(* IEC 61131-3 sources: AXOpen/src/showcase/app/src/core/AXOpen.AxoTask, 4 files *)

(* ---- AxoTaskAbortedExample.st ---- *)
USING AXOpen.Core;

NAMESPACE AxoTaskExamples

    // Demonstrates the Aborted terminal state in AxoTaskView:
    //   - Invoke kicks the task into Busy.
    //   - After a fixed number of Execute cycles, Abort() transitions the
    //     task to Aborted (stop icon + Resume button appear in the view).
    //   - Resume returns the task to Busy; counter is reset on Abort so the
    //     next run gets a fresh window before re-aborting.
    //   - Restore (Reset task button) returns the task to Ready.
    {S7.extern=ReadWrite}
    CLASS AxoTaskAbortedExample EXTENDS AXOpen.Core.AxoObject

        //<ComponentDeclaration>
        VAR PUBLIC
            {#ix-set:AttributeName = "<#Aborting task#>"}
            _abortingTask : AXOpen.Core.AxoTask;
            _counter : ULINT;
        END_VAR
        //</ComponentDeclaration>

        METHOD PUBLIC Execute

            //<Initialization>
            _abortingTask.Run(THIS);
            //</Initialization>

            //<AxoTaskAbortedPattern>
            IF _abortingTask.Execute() THEN
                _counter := _counter + ULINT#1;
                IF _counter > ULINT#250 THEN
                    _counter := ULINT#0;
                    _abortingTask.Abort();
                END_IF;
            END_IF;

            IF _abortingTask.IsReady() THEN
                _counter := ULINT#0;
            END_IF;
            //</AxoTaskAbortedPattern>

        END_METHOD
    END_CLASS
END_NAMESPACE

(* ---- AxoTaskDisabledExample.st ---- *)
USING AXOpen.Core;

NAMESPACE AxoTaskExamples

    // Demonstrates the disabled-state indicator in AxoTaskView:
    //   - The task is kept perpetually Busy (self-invoked, never completed),
    //     so it always sits in an "active" state.
    //   - Rendering this task through a DISABLED / display-only AxoTaskView
    //     (Disable=true, e.g. the Status presentation) draws the activity
    //     circle with a lock icon INSIDE it, instead of replacing the circle.
    //   - Note: a task disabled on the PLC side via SetIsDisabled(TRUE) aborts
    //     while Busy (see AxoTaskLight.Execute), so the lock-inside-circle
    //     visual is a VIEW-level disable of a genuinely running task.
    {S7.extern=ReadWrite}
    CLASS AxoTaskDisabledExample EXTENDS AXOpen.Core.AxoObject

        //<ComponentDeclaration>
        VAR PUBLIC
            {#ix-set:AttributeName = "<#Always-active task — render display-only#>"}
            _activeTask : AXOpen.Core.AxoTask;
            {#ix-set:AttributeName = "<#Idle (Ready) task — render display-only#>"}
            _idleTask : AXOpen.Core.AxoTask;
        END_VAR
        //</ComponentDeclaration>

        METHOD PUBLIC Execute

            //<Initialization>
            _activeTask.Run(THIS);
            _idleTask.Run(THIS);
            //</Initialization>

            //<AxoTaskAlwaysActivePattern>
            // Execute() first (satisfies the cyclic-execute-called check), then
            // Invoke(). Invoke() only acts while the task is Ready, so once the
            // task is Busy it is a no-op and the task stays active indefinitely.
            _activeTask.Execute();
            _activeTask.Invoke();
            //</AxoTaskAlwaysActivePattern>

            //<AxoTaskIdlePattern>
            // _idleTask is wired into the object tree but never invoked, so it
            // stays in the Ready (not-busy) state. Rendered through a disabled
            // view it shows the lock inside the empty Ready circle.
            //</AxoTaskIdlePattern>

        END_METHOD
    END_CLASS
END_NAMESPACE

(* ---- AxoTaskDocuExample.st ---- *)
USING AXOpen.Core;

NAMESPACE AxoTaskExamples
    {S7.extern=ReadWrite}
    CLASS AxoTaskDocuExample EXTENDS  AXOpen.Core.AxoObject
        VAR PUBLIC
            {#ix-set:AttributeName = "<#Task name#>"}
            _myTask : AxoTask;
            _myCounter : ULINT;
        END_VAR

        METHOD PUBLIC Initialize
            // Initialization of the context needs to be called first
            // It does not need to be called cyclically, just once
            _myTask.Run(THIS);
        END_METHOD

        METHOD PUBLIC Execute
            _myTask.Run(THIS);
            // Cyclicall call of the Execute
            IF _myTask.Execute() THEN
                _myCounter := _myCounter + ULINT#1;
                _myTask.DoneWhen(_myCounter = ULINT#100);
            END_IF;
            IF _myTask.IsDone() THEN
                _myCounter := ULINT#0;
            END_IF;
        END_METHOD

        METHOD Examples
        //<AxoTaskInvokeDone>
            IF _myTask.Invoke().IsDone() THEN
                ; //Do something
            END_IF;
        //</AxoTaskInvokeDone>

        //<AxoTaskInvokeDoneSeparatelly>
            _myTask.Invoke();

            IF _myTask.IsDone() THEN
                ; //Do something
            END_IF;
        //</AxoTaskInvokeDoneSeparatelly>

        //<AxoTaskRunning>
             IF _myTask.Invoke().IsBusy() THEN
                ; //Do something
            END_IF;
        //</AxoTaskRunning>

        //<AxoTaskError>
            IF _myTask.Invoke().HasError() THEN
                ; //Do something
            END_IF;
        //</AxoTaskError>

        //<AxoTaskInvoke>
            _myTask.Invoke();
        //</AxoTaskInvoke>
        END_METHOD
    END_CLASS

    //<AxoTaskEventLikeMethods>
    {S7.extern=ReadWrite}
    CLASS MyTaskExample EXTENDS AXOpen.Core.AxoTask
        VAR
            OnAbortCounter : ULINT;
            OnResumeCounter : ULINT;
            OnDoneCounter : ULINT;
            OnErrorCounter : ULINT;
            OnRestoreCounter : ULINT;
            OnStartCounter : ULINT;
            WhileErrorCounter : ULINT;
        END_VAR
        METHOD PROTECTED OVERRIDE OnAbort
            OnAbortCounter := OnAbortCounter + ULINT#1;
        END_METHOD

        METHOD PROTECTED OVERRIDE OnResume
            OnResumeCounter := OnResumeCounter + ULINT#1;
        END_METHOD

        METHOD PROTECTED OVERRIDE OnDone
            OnDoneCounter := OnDoneCounter + ULINT#1;
        END_METHOD

        METHOD PROTECTED OVERRIDE OnError
            OnErrorCounter := OnErrorCounter + ULINT#1;
        END_METHOD

        METHOD PROTECTED OVERRIDE OnRestore
            OnRestoreCounter := OnRestoreCounter + ULINT#1;
        END_METHOD

        METHOD PROTECTED OVERRIDE OnStart
            OnStartCounter := OnStartCounter + ULINT#1;
        END_METHOD

        METHOD PROTECTED OVERRIDE WhileError
            WhileErrorCounter := WhileErrorCounter + ULINT#1;
        END_METHOD
    END_CLASS
    //</AxoTaskEventLikeMethods>
END_NAMESPACE

(* ---- AxoTaskErrorExample.st ---- *)
USING AXOpen.Core;

NAMESPACE AxoTaskExamples

    // Demonstrates the Error terminal state in AxoTaskView:
    //   - Invoke kicks the task into Busy.
    //   - After a fixed number of Execute cycles, ErrorDetails is populated
    //     and ThrowWhen(TRUE) transitions the task to Error.
    //   - Restore (Reset task button) returns the task to Ready and clears
    //     the counter for the next demonstration.
    {S7.extern=ReadWrite}
    CLASS AxoTaskErrorExample EXTENDS AXOpen.Core.AxoObject

        //<ComponentDeclaration>
        VAR PUBLIC
            {#ix-set:AttributeName = "<#Failing task#>"}
            _failingTask : AXOpen.Core.AxoTask;
            _counter : ULINT;
        END_VAR
        //</ComponentDeclaration>

        METHOD PUBLIC Execute

            //<Initialization>
            _failingTask.Run(THIS);
            //</Initialization>

            //<AxoTaskErrorPattern>
            IF _failingTask.Execute() THEN
                _counter := _counter + ULINT#1;
                IF _counter > ULINT#250 THEN
                    _failingTask.ErrorDetails := 'Counter limit exceeded during execution.';
                    _failingTask.ThrowWhen(TRUE);
                END_IF;
            END_IF;

            IF _failingTask.IsReady() THEN
                _counter := ULINT#0;
            END_IF;
            //</AxoTaskErrorPattern>

        END_METHOD
    END_CLASS
END_NAMESPACE
